(* This function Block interfaces with a NO turbo valve*)
(* Mainly used in the FEE HXR GATT*)
FUNCTION F_TurboExtILK_NO : BOOL
VAR_INPUT
	Turbo		:	ST_PTM;
	BackingGauge:	ST_VG;
	InletGauge	:	ST_VG;
	VentValve	:	ST_VCC_NO; //NO type turbo valve
	ScrollPump	:	ST_RoughPump;
	Timer :TON;
END_VAR

VAR
END_VAR
VAR // added by the converter: edge detectors and wires of the graphical bodies
    _w1 : BOOL;
END_VAR

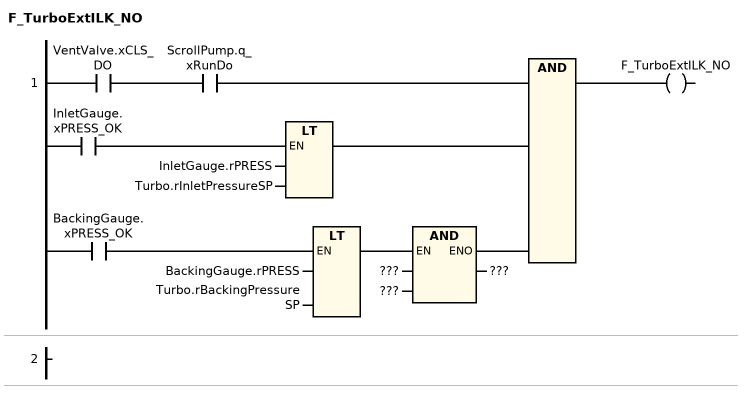
// NETWORK 1
_w1 := BackingGauge.xPRESS_OK AND BackingGauge.rPRESS < Turbo.rBackingPressureSP;
IF _w1 THEN (* ??? AND ???; result not used *) END_IF
F_TurboExtILK_NO := (VentValve.xCLS_DO AND ScrollPump.q_xRunDo) AND (InletGauge.xPRESS_OK AND InletGauge.rPRESS < Turbo.rInletPressureSP) AND _w1;

// NETWORK 2

END_FUNCTION

(* stored: Version 1.1.0.1, ProductVersion 3.1.4024.3
   POU F_TurboExtILK_NO: Id {3f22491e-9c00-45b3-979a-0a023cc045c2}, SpecialFunc None *)
